INTERFACE ITmsMover EXTENDS IMover

METHOD SetTrackId : BOOL
VAR_INPUT
	ActiveTrack : OTCID;
END_VAR
END_METHOD

END_INTERFACE

(* stored: Version 1.1.0.1, ProductVersion 3.1.4024.11
   Itf ITmsMover: Id {1dd4f0e1-1fa2-4d8b-bd4e-d91c7c33d591}
   Method SetTrackId: Id {6e62ed33-5211-41f4-b2cf-01546af65477} *)
